# EPICS autosave request: CARSApp/Db/XRMAnalyzer.req
$(P)$(Q):h
$(P)$(Q):k
$(P)$(Q):l
$(P)$(Q):dspace
$(P)$(Q):diam
$(P)$(Q):xtal
$(P)$(Q):Energy
$(P)$(Q):theta
$(P)$(Q):ana_dist
$(P)$(Q):det_x
$(P)$(Q):det_y
$(P)$(Q):det_track
$(P)$(Q):sim_mode
